Fanuc TP program (LS listing): h2_start.ls

/PROG  H2_START
/ATTR
OWNER		= MNEDITOR;
COMMENT		= "";
PROG_SIZE	= 384;
CREATE		= DATE 19-04-09  TIME 08:22:50;
MODIFIED	= DATE 19-04-16  TIME 11:21:48;
FILE_NAME	= H1_START;
VERSION		= 0;
LINE_COUNT	= 14;
MEMORY_SIZE	= 864;
PROTECT		= READ_WRITE;
TCD:  STACK_SIZE	= 0,
      TASK_PRIORITY	= 50,
      TIME_SLICE	= 0,
      BUSY_LAMP_OFF	= 0,
      ABORT_REQUEST	= 0,
      PAUSE_REQUEST	= 0;
DEFAULT_GROUP	= 1,*,*,*,*;
CONTROL_CODE	= 00000000 00000000;
/APPL
/MN
   1:  DO[29:HEATER2_START]=PULSE,1.0sec ;
   2:  WAIT   2.00(sec) ;
   3:   ;
   4:  //$WAITTMOUT=200 ;
   5:  //WAIT (DI[48:W1_DOOR_CLOSED]) TIMEOUT,LBL[1] ;
   6:   ;
   7:   ;
   8:  END ;
   9:  LBL[1] ;
  10:  MESSAGE[...] ;
  11:  MESSAGE[VRATA STROJA 1] ;
  12:  MESSAGE[NISU ZATVORENA] ;
  13:  WAIT (DI[48:W1_DOOR_CLOSED])    ;
  14:  END ;
/POS
/END
